Staubli VAL3: test.pjx

--- test.pjx ---
Parameters version=s7.11.2 stackSize=5000 millimeterUnit=true
Program file=start.pgx
Program file=stop.pgx
Data file=test.dtx

--- test.dtx ---
mdesc mNomSpeed
tool tTool = {fatherId=flange[0], ioLink=valve1}
jointRx jAproachPiece = {j1=-5.03067209967487, j2=43.3081121684082, j3=54.1351709463615, j4=4.70507356684578, j5=79.1734286699559, j6=-42.7327028817804}
jointRx jHome
pointRx pGetObject = {x=535.804523528443, y=9.14837989701774, z=-274.924299394303, rx=4.31323960308358, ry=176.199656586078, rz=-37.0974828689112, fatherId=world[0]}

--- start.pgx ---
program start()
begin
  movej(jHome,tTool,mNomSpeed)
  waitEndMove()
  movej(jAproachPiece,tTool,mNomSpeed)
  waitEndMove()
  movel(pGetObject,tTool,mNomSpeed)
  waitEndMove()
  open()
  waitEndMove()
  movej(jAproachPiece,tTool,mNomSpeed)
  waitEndMove()

end
